# EPICS substitutions: siteApps/WinShmIOC/ioctestApp/Db/user.substitutions
# Example substitutions file

file "db/circle.db" {
    { user = "silee" }
}

file "db/dbExample1.db" {
    { user = "silee" }
}

file db/dbExample2.db {
    pattern { user, no, scan }
        { "silee", 1, "1 second" }
        { "silee", 2, "2 second" }
        { "silee", 3, "5 second" }
}
